FUNCTION_BLOCK AND_3 (* FB to calculate bitwise boolean AND (generic FB) *)
  (* Standard: 61499-1 *)
  (* Version 1.0, 2014-10-11, Matthias Plasch, 4DIAC-Consortium, matthias.plasch@profactor.at *)
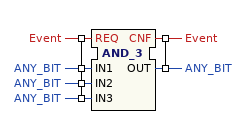
  EVENT_INPUT
    REQ WITH IN1, IN2, IN3; (* Normal Execution Request *)
  END_EVENT
  EVENT_OUTPUT
    CNF WITH OUT; (* Execution Confirmation *)
  END_EVENT
  VAR_INPUT
    IN1 : ANY_BIT; (* AND input 1 *)
    IN2 : ANY_BIT; (* AND input 2 *)
    IN3 : ANY_BIT; (* AND input 3 *)
  END_VAR
  VAR_OUTPUT
    OUT : ANY_BIT; (* AND result *)
  END_VAR
END_FUNCTION_BLOCK
